% RSLogix 500 project Ladder_Identificacion_Presion.RSS, saved by version 7.30.00.17 %
PROJECT "UNTITLED"    % processor: MicroLogix 1500 %

PROGRAM FILES
  LAD 2   3 rungs

DATA FILES
  O0 OUTPUT  6 elements
  I1 INPUT  12 elements
  S2 STATUS  66 elements
  B3 BINARY  1 elements
  T4 TIMER  1 elements
  C5 COUNTER  1 elements
  R6 CONTROL  1 elements
  N7 INTEGER  10 elements
  F8 FLOAT  1 elements

LADDER 2
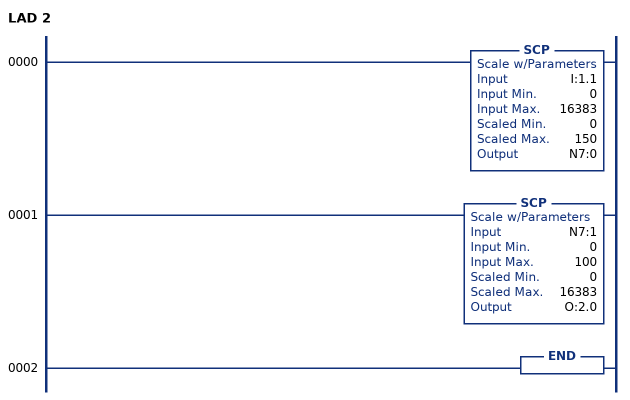
% Rung: 0 %
SOR SCP I:1.1 0 16383 0 150 N7:0 EOR
% Rung: 1 %
SOR SCP N7:1 0 100 0 16383 O:2.0 EOR
% Rung: 2 %
SOR END EOR

OTHER DOCUMENTED ADDRESSES
  I:1.0  N
